FUNCTION_BLOCK fb_XmlWrite
VAR_INPUT
  bExecute      : BOOL;
  sFilePath     : STRING(255);(*File and Path Name*)
  sXPath        : STRING;     (*Dataentry in XML file*)
  pData         : pvoid;      (*pointer to Datafield*)
  diSize        : UDINT;      (*size of datafield*)
END_VAR
VAR_OUTPUT
  bBusy         : BOOL;
  bDone         : BOOL;
  bError        : BOOL;
  nError        : UDINT;
END_VAR
VAR
  rtrigIn       : Tc2_Standard.R_TRIG;
  ftrigIn       : Tc2_Standard.F_TRIG;
  diStep        : DINT;
  sMsg          : ARRAY[1..10] OF STRING;
  iMsg          : DINT := 1;

  fbWriteData   : Tc2_XmlDataSrv.FB_XmlSrvWrite;
END_VAR


rtrigIn(CLK:= bExecute);
ftrigIn(CLK:= bExecute);


IF rtrigIn.Q
THEN
  bBusy := TRUE;
  bDone := FALSE;
  bError:= FALSE;
  diStep  := 10;
END_IF

IF ftrigIn.Q
THEN
  fbWriteData(bExecute := FALSE);
  diStep  := 0;
END_IF

CASE diStep OF

  0:
    bBusy := FALSE;
    bDone := FALSE;
    bError:= FALSE;

  10:
    sMsg[iMsg] := 'start: ';
    iMsg := iMsg + 1;
    fbWriteData(bExecute := FALSE);
    diStep := 15;

  15:
    fbWriteData(
      bExecute := TRUE,
      sNetId:= '', 
      ePath       := PATH_GENERIC, 
      nMode       := Tc2_XmlDataSrv.XMLSRV_ADDMISSING, 
      pSymAddr    := pData, 
      cbSymSize   := diSize, 
      sFilePath   := sFilePath, 
      sXPath      := sXPath, 
      bExecute:= , 
      tTimeout    := T#5S, 
      bBusy=> , 
      bError=> , 
      nErrId=> );

    IF fbWriteData.bBusy
    THEN
      sMsg[iMsg] := 'busy: ';
      iMsg := iMsg + 1;
      diStep := 20;
    END_IF

  20:
    fbWriteData();
    IF NOT fbWriteData.bError
    THEN
      nError := 0;
      IF NOT fbWriteData.bBusy
      THEN
        sMsg[iMsg] := 'done: ';
        iMsg := iMsg + 1;
        fbWriteData(bExecute := FALSE);
        diStep := 30;
      END_IF
    ELSE
      IF fbWriteData.nErrId <> 0
      THEN
        nError := fbWriteData.nErrId;
        sMsg[iMsg] := 'error: ';
        sMsg[iMsg] := concat(sMsg[iMsg], TO_STRING(fbWriteData.nErrId));
        iMsg := iMsg + 1;

        fbWriteData(bExecute := FALSE);
        diStep := 99;
      END_IF
    END_IF

  30:
    bBusy := FALSE;
    bDone := TRUE;

  99:
    bBusy  := FALSE;
    bError := TRUE;
END_CASE

IF (iMsg > 10) THEN iMsg :=1; END_IF

END_FUNCTION_BLOCK

(* stored: Version 1.1.0.1, ProductVersion 3.1.4026.20
   POU fb_XmlWrite: Id {518bf6cd-fb6b-4abd-8df3-fa1a2b9c3532}, SpecialFunc None *)
